FUNCTION llenadoTanque : BOOL
VAR_INPUT
END_VAR
VAR
END_VAR

END_FUNCTION

(* stored: Version 1.1.0.1, ProductVersion 3.1.4024.15
   POU llenadoTanque: Id {730c9376-bdb9-48a0-bb3c-62f695fd5010}, SpecialFunc None *)
